FUNCTION_BLOCK TrackingBlock
VAR_INPUT
	
	fbMotorReference : REFERENCE TO FB_AnalogMotorDriver;
	fbMetadata : REFERENCE TO MetadataBlock; 

END_VAR
VAR_OUTPUT
	
	nEncoderCounts : LINT; 
	rEncoderDegrees : REAL;
	rEncoderLastDegrees : REAL;
	rEncoderRadians : REAL; 
	rEncoderLastRadians : REAL;
	rEncoderRadiansBuffer : ARRAY[1..FILTER_WINDOW] OF REAL;
	rEncoderRadiansSum : REAL;
	rEncoderRadiansFiltered : REAL;
	nFilterBufferCount : INT := 0;
	rGripForce : REAL;

END_VAR
VAR
	
	fbEncoder1 : FB_QuadratureEncoder; 
	fbLoadCell : FB_AnalogLoadCellInput; 
	i : INT;
	j : INT;
	z : LINT := 0; 

END_VAR
VAR CONSTANT
	FILTER_WINDOW : INT := 11;
END_VAR

///////////// Read sensors on current iteration
// Encoders 
fbEncoder1(); 
nEncoderCounts := fbEncoder1.nNetCounts; 
rEncoderDegrees := fbEncoder1.rDegrees; 
rEncoderLastDegrees := fbEncoder1.rLastDegrees; 
rEncoderRadians := fbEncoder1.rRadians; 
rEncoderLastRadians := fbEncoder1.rLastRadians; 

// test
z := z + 1;

// Update digital filter. 
IF nFilterBufferCount < FILTER_WINDOW THEN 
	nFilterBufferCount := nFilterBufferCount + 1; 
END_IF

// Shift the buffer and add the new reading 
FOR i := FILTER_WINDOW TO 2 BY -1 DO
	rEncoderRadiansBuffer[i] := rEncoderRadiansBuffer[i-1]; 
END_FOR
rEncoderRadiansBuffer[1] := rEncoderRadians;

// Computer the moving average only if the buffer is full
j := MIN(nFilterBufferCount, FILTER_WINDOW); 
rEncoderRadiansSum := 0.0; 
FOR i:= 1 TO j DO
	rEncoderRadiansSum := rEncoderRadiansSum + rEncoderRadiansBuffer[i];
END_FOR
rEncoderRadiansFiltered := rEncoderRadiansSum / j; 

// Load cell 
fbLoadCell(); 
rGripForce := fbLoadCell.rCalibratedOutput; 
///////////// End sensor reading 

//////////////// Report back to main 
GVL.ENCODER_1_COUNTER_VALUE := nEncoderCounts; 
GVL.ENCODER_1_DEGREES := rEncoderDegrees; 
GVL.LOAD_CELL_NEWTONS := rGripForce;

METHOD Reset : BOOL
VAR_INPUT
END_VAR
fbEncoder1.Reset();
END_METHOD

END_FUNCTION_BLOCK

(* stored: Version 1.1.0.1, ProductVersion 3.1.4024.12
   POU TrackingBlock: Id {b0575d33-e51d-481f-8c5c-542abf7c6b2e}, SpecialFunc None
   Method Reset: Id {ce4aa878-021e-4bf9-b715-d2c076cdb3a8} *)
